SUBAPPLICATION Versuch_409 (* Versuch Array Summe *)
  (* Standard: 61499-2; Description: Copyright (c) 2023 Meisterschulen am Ostbahnhof This program and the accompanying materials are made available under the terms of the Eclipse Public License 2.0 which is available at https://www.eclipse.org/legal/epl-2.0/ SPDX-License-Identifier: EPL-2.0 *)
  (* Version 1.0, 2023-10-23, Franz Höpfinger, Meisterschulen am Ostbahnhof *)
  PACKAGE Versuche;
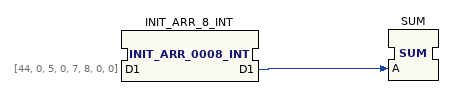
  FBS
    SUM : logiBUS::utils::dyn_arr::SUM;
    INIT_ARR_8_INT : logiBUS::utils::generate::INIT_ARR_0008_INT(D1 := [44, 0, 5, 0, 7, 8, 0, 0]);
  END_FBS
  DATA_CONNECTIONS
    INIT_ARR_8_INT.D1 TO SUM.A;
  END_CONNECTIONS
END_SUBAPPLICATION
